FUNCTION_BLOCK interResourceRxLReal (* goFB_ignore *)
  (* Standard: 61499-2 *)
  (* Version 0.1, 2017-00-25, hpea485, UOA *)
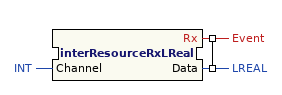
  EVENT_OUTPUT
    Rx WITH Data;
  END_EVENT
  VAR_INPUT
    Channel : INT;
  END_VAR
  VAR_OUTPUT
    Data : LREAL;
  END_VAR
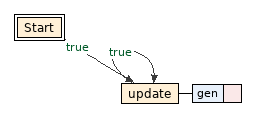
  EC_STATES
    Start;
    update : gen;
  END_STATES
  EC_TRANSITIONS
    Start TO update := true;
    update TO update := true;
  END_TRANSITIONS
  ALGORITHM gen IN C:
if(something) {
	something;
	something;
	me->outputEvents.Rx = 1;
}
  END_ALGORITHM
END_FUNCTION_BLOCK
